// TIA Portal V19 export
DATA_BLOCK "DO MAPING"   // DB2
{ S7_Optimized_Access := 'TRUE' }
// stored: MemoryReserve 100
   VAR
      "HOOTER-1" : Bool;
      "HOOTER-2" : Bool;
      "MFG VESSEL MOTOR" : Bool;
      "PREMIXING VESSEL MOTOR" : Bool;
      "STORAGE VESSEL-1 MOTOR" : Bool;
      "STORAGE VESSEL-2 MOTOR" : Bool;
      "INLINE HOMOGENIZER-1" : Bool;
      "FILTER PRESS MOTOR" : Bool;
      "INLINE HOMOGENIZER-2" : Bool;
      "MFG LOBE PUMP" : Bool;
      "STORAGE VESSEL-1 LOBE PUMP" : Bool;
      "STORAGE VESSEL-2 LOBE PUMP" : Bool;
      "SUGAR VESSEL MOTOR" : Bool;
      "BASKET FILTER MOTOR" : Bool;
      "VACUUME PUMP-1" : Bool;
      "VACUUME PUMP-2" : Bool;
      "CIP FORWARD PUMP" : Bool;
      "CIP REVERSE PUMP" : Bool;
      "DOSING PUMP-1 ALKALI" : Bool;
      "DOSING PUMP-2 ACID" : Bool;
      "MFG VESSEL LAMP" : Bool;
      "PREMIXING VESSEL LAMP" : Bool;
      "STORAGE VESSEL-1 LAMP" : Bool;
      "STORAGE VESSEL-2 LAMP" : Bool;
      "SUGAR VESSEL LAMP" : Bool;
      "PBV-01 ON SUGAR SUCTION LINE" : Bool;
      "PBV- 02 ON VACUUM INLET LINE" : Bool;
      "PBV- 03 ON VENT FILTER" : Bool;
      "PAV- 03 ON AIR INLET LINE" : Bool;
      "PBV- 04 FROM BOTTOM OUTLET TO CIP INLET LINE" : Bool;
      "PBV- 05 ON SPRAY BALL INLET LINE" : Bool;
      "PBV- 06 ON PW INLET LINE" : Bool;
      "PBV- 07 ON VACUUM VENT LINE" : Bool;
      "PAV- 07 ON SEAL COOLING INLET LINE FOR STIRRER" : Bool;
      "PAV- 08 ON AIR INLET LINE" : Bool;
      "PAV- 09 ON STEAM INLET LINE" : Bool;
      "PAV- 10 ON STEAM OUTLET LINE" : Bool;
      "PAV- 11 ON SEAL COOLING INLET LINE" : Bool;
      "PBV- 12 FROM BOTTOM OUTLET TO CIP DRAIN LINE" : Bool;
      "PBV- 13 FROM BOTTOM OUTLET TO CIP INLET LINE" : Bool;
      "PBV- 14 ON BOTTOM OUTLET LINE" : Bool;
      "PBV- 15 FROM BOTTOM OUTLET TO DRAIN LINE" : Bool;
      "PBV- 16 FROM BOTTOM OUTLET TO BASKET FILTER INLET LINE" : Bool;
      "PBV- 17 ON BASKET FILTER INLET LINE" : Bool;
      "PBV- 18 ON BASKET FILTER OUTLET LINE" : Bool;
      "PBV- 19 ON SUGAR VESSEL CIP INLET LINE" : Bool;
      "PBV- 20 ON PREMIXING VESEL CIP INLET LINE" : Bool;
      "PBV- 21 ON PW INLET BYPASS LINE" : Bool;
      "PBV- 22 ON PW INLET LINE" : Bool;
      "PBV- 23 ON VENT FILTER" : Bool;
      "PBV- 24 ON VACUUM INLET LINE" : Bool;
      "PBV- 25 FROM BOTTOM OUTLET TO SPRAY BALL INLET LINE" : Bool;
      "PBV- 26 ON SPRAY BALL INLET LINE" : Bool;
      "PBV- 27 FROM SUGAR TO PREMIXING VESSEL INLET LINE" : Bool;
      "PBV- 28 ON VESSEL TOP DISH" : Bool;
      "PBV- 29 ON RECIRCULATION LINE" : Bool;
      "PBV- 30 FROM PREMIXING TO STORAGE TRANSFER LINE" : Bool;
      "PBV- 31 FROM SORBITOL VESSEL TO PREMIXING VESSEL TRANSFER LINE" : Bool;
      "PBV- 32 FROM PREMIXING TO MFG TRANSFER LINE" : Bool;
      "PAV- 33 ON STEAM INLET LINE" : Bool;
      "PAV- 35 ON COOLING WATER OUTLET LINE" : Bool;
      "PAV- 36 ON STEAM OUTLET LINE" : Bool;
      "PAV- 37 ON BYPASS CONDENSATE LINE" : Bool;
      "PAV- 38 ON COOLING WATER INLET LINE" : Bool;
      "PBV- 39 FROM BOTTOM OUTLET TO SPRAY BALL INLET LINE" : Bool;
      "PBV- 40 FROM BOTTOM OUTLET TO SPRAY BALL INLET LINE" : Bool;
      "PBV- 41 FROM BOTTOM OUTLET TO DRAIN LINE" : Bool;
      "PBV- 42 FROM BOTTOM OUTLET TO DRAIN LINE" : Bool;
      "PBV- 43 FROM BOTTOM OUTLET TO INLINE HOMOGENIZER LINE" : Bool;
      "PBV- 44 FROM VESSEL OUTLET TO FILTER PRESS LINE" : Bool;
      "PBV- 45 FROM INLINE HOMOGENIZER TO STORAGE TRANSFER LINE" : Bool;
      "PBV- 46 ON INLINE HOMOGENIZER INLET LINE" : Bool;
      "PBV- 47 ON INLINE HOMOGENIZER RECIRCULATION LINE" : Bool;
      "PAV- 48 ON SEAL COOLING INLET LINE FOR INLINE HOMOGENIZER" : Bool;
      "PBV- 49 INLINE HOMOGENIZER DRAIN LINE" : Bool;
      "PBV- 50 ON PW INLET LINE" : Bool;
      "PBV- 51 FROM PW INLET TO DRAIN LINE" : Bool;
      "PBV- 52 FROM SUGAR MELTING TO MFG VESSEL TRANSFER LINE" : Bool;
      "PBV- 53 ON VENT FILTER" : Bool;
      "PBV- 54 FROM BOTTOM OUTLET TO SPRAY BALL INLET LINE" : Bool;
      "PBV- 55 ON SPRAY BALL INLET LINE" : Bool;
      "PBV- 56 ON VACUUM INLET LINE" : Bool;
      "PBV- 57 ON RECIRCULATION LINE" : Bool;
      "PBV- 58 FROM INLINE HOMOGENIZER TO STORAGE TRANSFER LINE" : Bool;
      "PBV- 59 FROM PREMIXING TO FILTER PRESS TRANSFER LINE" : Bool;
      "PBV- 60 FROM PREMIXING LOBE PUMP TO FILTER PRESS LINE" : Bool;
      "PAV- 61 ON COOLING OUTLET LINE" : Bool;
      "PAV- 62 ON STEAM INLET LINE" : Bool;
      "PAV- 63 ON COOLING INLET LINE" : Bool;
      "PAV- 64 ON SEAL COOLING INLET LINE FOR STIRRER" : Bool;
      "PAV- 65 ON STEAM OUTLET LINE" : Bool;
      "PAV- 66 ON BYPASS CONDENSATE LINE" : Bool;
      "PBV- 67 FROM BOTTOM OUTLET TO SPRAY BALL INLET LINE" : Bool;
      "PBV- 68 FROM BOTTOM OUTLET TO SPRAY BALL INLET LINE" : Bool;
      "PBV- 69 FROM BOTTOM OUTLET TO DRAIN LINE" : Bool;
      "PBV- 70 FROM BOTTOM OUTLET TO DRAIN LINE" : Bool;
      "PBV- 71 FROM BOTTOM OUTLET TO INLINE HOMOGENIZER LINE" : Bool;
      "PBV- 72 ON INLINE HOMOGENIZER INLET LINE" : Bool;
      "PBV- 73 ON RECIRCULATION LINE" : Bool;
      "PBV- 74 FROM BOTTOM OUTLET TO INLINE HOMOGENIZER LINE" : Bool;
      "PAV- 75 ON SEAL COOLING INLET LINE FOR HOMOGENIZER" : Bool;
      "PBV- 76 FROM INLINE HOMOGENIZER TO DRAIN LINE" : Bool;
      "PBV- 77 ON FILTER PRESS INLET LINE" : Bool;
      "PBV- 78 ON FILTER PRESS OUTLET LINE" : Bool;
      "PBV- 79 ON FILTER PRESS OUTLET LINE" : Bool;
      "PBV- 80 FROM MFG TO STORAGE VESSEL TRANSFER LINE" : Bool;
      "PBV- 81 ON VESSEL TOP DISH" : Bool;
      "PBV- 82 FROM BOTTOM OUTLET TO SPRAY BALL INLET LINE" : Bool;
      "PBV- 83 ON CIP INLET LINE" : Bool;
      "PAV- 84 ON SEAL COOLING LINE OF BOTTOM STIRRER" : Bool;
      "PBV- 85 FROM BOTTOM OUTLET TO SPRAY BALL INLET LINE" : Bool;
      "PBV- 86 FROM BOTTOM OUTLET TO DRAIN LINE" : Bool;
      "PBV- 87 FROM BOTTOM OUTLET TO SPRAY BALL INLET LINE" : Bool;
      "PBV- 88 FROM BOTTOM OUTLET TO DRAIN LINE" : Bool;
      "PBV- 89 FROM VESSEL BOTTOM OUTLET TO LOBE PUMP LINE" : Bool;
      "PBV- 90 ON VESSEL TOP DISH" : Bool;
      "PBV- 91 FROM BOTTOM OUTLET TO SPRAY BALL INLET LINE" : Bool;
      "PBV- 92 ON SPRAY BALL INLET LINE" : Bool;
      "PAV- 93 ON SEAL COOLING LINE OF BOTTOM STIRRER" : Bool;
      "PBV- 94 FROM BOTTOM OUTLET TO SPRAY BALL INLET LINE" : Bool;
      "PBV- 95 FROM BOTTOM OUTLET TO DRAIN LINE" : Bool;
      "PBV- 96 FROM BOTTOM OUTLET TO SPRAY BALL INLET LINE" : Bool;
      "PBV- 97 FROM BOTTOM OUTLET TO DRAIN LINE" : Bool;
      "PBV- 98 FROM BOTTOM OUTLET TO LOBE PUMP LINE" : Bool;
      "PBV- 99 ON VACUUM VENT LINE" : Bool;
      "PFBV- 100 ON VESSEL BOTTOM DISH" : Bool;
      "PFBV- 101 ON VESSEL BOTTOM DISH" : Bool;
      "PFBV- 102 ON VESSEL BOTTOM DISH" : Bool;
      "PFBV- 103 ON VESSEL BOTTOM DISH" : Bool;
      "PFBV- 104 ON VESSEL BOTTOM DISH" : Bool;
      "PAV- 105 ON AIR INLET LINE" : Bool;
      "SPARE-1" : Bool;
      "SPARE-2" : Bool;
      "SPARE-3" : Bool;
      "SPARE-4" : Bool;
      "SPARE-5" : Bool;
      "SPARE-6" : Bool;
      "SPARE-7" : Bool;
      "SPARE-8" : Bool;
      "SPARE-9" : Bool;
      "SPARE-10" : Bool;
      "SPARE-11" : Bool;
      "SPARE-12" : Bool;
      "SPARE-13" : Bool;
      "SPARE-14" : Bool;
      "SPARE-15" : Bool;
      "SPARE-16" : Bool;
      "SPARE-17" : Bool;
      "SPARE-18" : Bool;
      "SPARE-19" : Bool;
      "SPARE-20" : Bool;
      "SPARE-21" : Bool;
      "SPARE-22" : Bool;
      "SPARE-23" : Bool;
      "SPARE-24" : Bool;
      "SPARE-25" : Bool;
      "SPARE-26" : Bool;
      "SPARE-27" : Bool;
      "SPARE-28" : Bool;
      "SPARE-29" : Bool;
      "SPARE-30" : Bool;
      "SPARE-31" : Bool;
      "SPARE-32" : Bool;
      "SPARE-33" : Bool;
      "SPARE-34" : Bool;
      "SPARE-35" : Bool;
      "SPARE-36" : Bool;
      "SPARE-37" : Bool;
      "SPARE-38" : Bool;
      "SPARE-39" : Bool;
      "SPARE-40" : Bool;
      "SPARE-41" : Bool;
      "SPARE-42" : Bool;
      "SPARE-43" : Bool;
      "SPARE-44" : Bool;
      "SPARE-45" : Bool;
   END_VAR
BEGIN
END_DATA_BLOCK
